// TIA Portal V17 export
// export: Created 2025-03-05T08:01:54.8682733Z, ExportSetting WithDefaults, DisplayName Totally Integrated Automation Portal, DisplayVersion V17 Update 8, DisplayName TIA Portal Openness, DisplayVersion V17 Update 8, DisplayName TIA Portal Version Control Interface, DisplayVersion V17, DisplayName SINAMICS Startdrive Advanced, DisplayVersion V17 SP2, DisplayName SINAMICS Startdrive G110M, G120, G120C, G120D, G120P, G115D, DisplayVersion V17 SP2, DisplayName SINAMICS Startdrive G130, G150, S120, S150, SINAMICS MV, S210, DisplayVersion V17 SP2, DisplayName STEP 7 Professional, DisplayVersion V17 Update 8, DisplayName SINUMERIK ONE STEP 7 Toolbox, DisplayVersion V17 Update 12, DisplayName SINUMERIK 840D sl STEP 7 Toolbox, DisplayVersion V17 Update 12, DisplayName STEP 7 Safety, DisplayVersion V17 Update 6, DisplayName WinCC Advanced, DisplayVersion V17 Update 8
TYPE "LBP_typeHMI"
TITLE = Operator panel signals / Señales panel de mando / Bedienfeld-Signale
// User data type for block LBP_HMI [DB19] / Tipo de dato de usuario para bloque LBP_HMI [DB19] / Anwender-Datentyp für Baustein LBP_HMI [DB19]
// stored: IsFailsafeCompliant false
   STRUCT
      A_SCLight : Bool;   // Bildschirm hell / Screen light / Pantalla luminosa
      A_SCDark : Bool;   // Bildschirm Abdunkelung / Screen darkening / Atenuación pantalla
      A_KeyDisable : Bool;   // Taste deaktivieren / Key disable / Desactivar tecla
      A_ClearCanAl : Bool;   // Abbruch-Alarme löschen / Clear cancel alarms / Borrar alarmas de cancelación
      A_ClearRecAl : Bool;   // Rückruf-Alarme löschen / Clear recall alarms / Borrar alarmas de rellamada
      f0_5 : Bool;
      A_SafeActionLog : Bool;   // Flankenwechsel 0 → 1: ACTION.COM nach CRASH.COM speichern / Edge change 0 → 1: Save ACTION.COM to CRASH.COM / Cambio de flanco 0 → 1: guardar ACTION.COM a CRASH.COM
      A_ActWCS : Bool;   // Istwert in WCS 0=MCS / Actual value in WCS 0=MCS / Valor real en WCS 0=MCS
      A_PLCExtViewerReject : Bool;   // Externen Viewer ablehnen / External viewer reject / Rechazar visualizador externo
      A_PLCExtViewerMode : Bool;   // Externer Viewer-Modus / External viewer mode / Modo de visualizador externo
      f1_2 : Bool;
      f1_3 : Bool;
      f1_4 : Bool;
      f1_5 : Bool;
      f1_6 : Bool;
      f1_7 : Bool;
      A_1stError1 : Word;   // 1. Fehler HIGRAPH / 1st error HIGRAPH / 1.er error HIGRAPH
      A_1stError2 : Word;   // 1. Fehler HIGRAPH / 1st error HIGRAPH / 1.er error HIGRAPH
      A_ASpi1percent : Byte;   // Analogspindel 1: / Analog spindle 1: / Cabezal analógico 1:
      A_ASpi2percent : Byte;
      A_MCPChan : Byte;
      A_OEM1 : Bool;
      A_OEM2 : Bool;
      A_AToolMeas : Bool;   // AutoToolMeasure
      f9_3 : Bool;
      f9_4 : Bool;
      f9_5 : Bool;
      f9_6 : Bool;
      f9_7 : Bool;
      A_Hardkey : Byte;   // PLC Hardkeys / PLC hardkeys / Pulsadores de función PLC
      f11 : Byte;   // Reserviert für Hardkeys / Reserved for hardkeys / Reservado para pulsadores de función
      f12_0 : Bool;
      f12_1 : Bool;
      A_COM2 : Bool;
      A_COM1 : Bool;
      A_V24stop : Bool;
      A_V24ext : Bool;
      A_V24off : Bool;
      A_V24on : Bool;
      A_TeachDisable : Bool;
      f13_1 : Bool;
      f13_2 : Bool;
      f13_3 : Bool;
      f13_4 : Bool;
      A_PPdeload : Bool;
      A_PPload : Bool;
      A_PPsel : Bool;
      A_V24Index1 : Byte;
      A_V24Index2 : Byte;
      A_V24NoFile1 : Byte;
      A_V24NoFile2 : Byte;
      A_res18 : Byte;
      A_res19 : Byte;   // Meldungszähler / Message counter / Contador de avisos
      f20_0 : Bool;
      E_SCDark : Bool;   // Bildschirm Abdunkelung / Screen darkening / Atenuación pantalla
      E_Cancel : Bool;   // Abbruch / Cancel / Cancelación
      E_CanCleared : Bool;   // Abbruch-Alarme gelöscht / Cancel alarms cleared / Alarmas de cancelación borradas
      E_RecCleared : Bool;   // Rückruf-Alarme gelöscht / Recall alarms cleared / Alarmas de rellamada borradas
      f20_5 : Bool;   // res. Sprache / res. language / Lenguaje res.
      E_SimActiv : Bool;   // Simulation aktiv / Simulation active / Simulación activa
      E_ActWCS : Bool;   // Umschaltung MCS/WCS 0=MCS / Switchover MCS/WCS 0=MCS / Conmutación MCS/WCS 0=MCS
      E_ActivWA : Byte;
      E_Chan : Byte;   // Kanal angezeigt / Channel displayed / Canal mostrado
      E_KeybHandl : Bool;   // Tastatur Handhabung / Keyboard handling / Manejo del teclado
      E_DataTransf : Bool;   // Datenübertragung aktiv / Data transfer active / Transferencia de datos activa
      E_DisplChange : Bool;   // Display Änderung / Display change / Cambio de visualización
      f23_3 : Bool;
      f23_4 : Bool;
      f23_5 : Bool;
      f23_6 : Bool;
      f23_7 : Bool;
      E_ScreenNo : Word;
      E_res26_0 : Bool;   // Reserviert / Reserved / Reservado
      E_PPOK : Bool;   // Teileprogramm-Status OK / Part program status OK / Estado programa de pieza OK
      E_PPErr : Bool;   // Teileprogramm Statusfehler / Part program status error / Estado programa de pieza error
      E_PPAct : Bool;   // Teileprogramm-Status aktiv / Part program status active / Estado programa de pieza activo
      f26_4 : Bool;   // Reserviert / Reserved / Reservado
      E_PPdeload : Bool;   // Teileprogramm-Status wird entladen / Part program status deloading / Estado programa de pieza en descarga
      E_PPload : Bool;   // Teileprogramm-Status wird geladen / Part program status loading / Estado programa de pieza en carga
      E_PPsel : Bool;   // Teileprogramm-Status wird ausgewählt / Part program status selecting / Estado programa de pieza se selecciona
      E_PPError : Byte;   // Teileprogramm Statusfehler / Part program status error / Estado programa de pieza error
      A_PictNo : Int;
      A_PictOn : Bool;
      A_PictOff : Bool;
      f30_2 : Bool;
      f30_3 : Bool;
      f30_4 : Bool;
      f30_5 : Bool;
      f30_6 : Bool;
      f30_7 : Bool;
      E_PictOK : Bool;
      E_PictOn : Bool;
      E_PictAct : Bool;
      E_PictOff : Bool;
      E_PictErr : Bool;
      f31_5 : Bool;
      f31_6 : Bool;
      E_NotAct : Bool;
      A_FuncNo : Byte;
      A_Par1 : Byte;
      A_Par2 : Byte;
      A_Par3 : Byte;
      E_FuncErr : Byte;
      f37 : Byte;
      f38 : Byte;
      f39 : Byte;
      res40 : Array[0..9] of Byte;
      MMC2 : Struct
         A_SCLight : Bool;   // Bildschirm hell / Screen light / Pantalla luminosa
         A_SCDark : Bool;   // Bildschirm Abdunkelung / Screen darkening / Atenuación pantalla
         A_KeyDisable : Bool;   // Taste deaktivieren / Key disable / Desactivar tecla
         A_ClearCanAl : Bool;   // Abbruch-Alarme löschen / Clear cancel alarms / Borrar alarmas de cancelación
         A_ClearRecAl : Bool;   // Rückruf-Alarme löschen / Clear recall alarms / Borrar alarmas de rellamada
         f0_5 : Bool;
         f0_6 : Bool;
         A_ActWCS : Bool;   // Istwert in WCS 0=MCS / Actual value in WCS 0=MCS / Valor real en WCS 0=MCS
         A_PLCExtViewerReject : Bool;   // Externen Viewer ablehnen / External viewer reject / Rechazar visualizador externo
         A_PLCExtViewerMode : Bool;   // Externer Viewer-Modus / External viewer mode / Modo de visualizador externo
         f1_2 : Bool;
         f1_3 : Bool;
         f1_4 : Bool;
         f1_5 : Bool;
         f1_6 : Bool;
         f1_7 : Bool;
         A_1stError1 : Word;   // 1. Fehler HIGRAPH / 1st error HIGRAPH / 1.er error HIGRAPH
         A_1stError2 : Word;   // 1. Fehler HIGRAPH / 1st error HIGRAPH / 1.er error HIGRAPH
         A_ASpi1percent : Byte;   // Analogspindel 1: / Analog spindle 1: / Cabezal analógico 1:
         A_ASpi2percent : Byte;
         A_MCPChan : Byte;
         A_OEM1 : Bool;
         A_OEM2 : Bool;
         A_AToolMeas : Bool;   // AutoToolMeasure
         f9_3 : Bool;
         f9_4 : Bool;
         f9_5 : Bool;
         f9_6 : Bool;
         f9_7 : Bool;
         A_Hardkey : Byte;   // PLC Hardkeys / PLC hardkeys / Pulsadores de función PLC
         f11 : Byte;   // Reserviert für Hardkeys / Reserved for hardkeys / Reservado para pulsadores de función
         f12_0 : Bool;
         f12_1 : Bool;
         A_COM2 : Bool;
         A_COM1 : Bool;
         A_V24stop : Bool;
         A_V24ext : Bool;
         A_V24off : Bool;
         A_V24on : Bool;
         A_TeachDisable : Bool;
         f13_1 : Bool;
         f13_2 : Bool;
         f13_3 : Bool;
         f13_4 : Bool;
         A_PPdeload : Bool;
         A_PPload : Bool;
         A_PPsel : Bool;
         A_V24Index1 : Byte;
         A_V24Index2 : Byte;
         A_V24NoFile1 : Byte;
         A_V24NoFile2 : Byte;
         A_res18 : Byte;
         A_res19 : Byte;   // Meldungszähler / Message counter / Contador de avisos
         f20_0 : Bool;
         E_SCDark : Bool;   // Bildschirm Abdunkelung / Screen darkening / Atenuación pantalla
         E_Cancel : Bool;   // Abbruch / Cancel / Cancelación
         E_CanCleared : Bool;   // Abbruch-Alarme gelöscht / Cancel alarms cleared / Alarmas de cancelación borradas
         E_RecCleared : Bool;   // Rückruf-Alarme gelöscht / Recall alarms cleared / Alarmas de rellamada borradas
         f20_5 : Bool;   // res. Sprache / res. language / Lenguaje res.
         E_SimActiv : Bool;   // Simulation aktiv / Simulation active / Simulación activa
         E_ActWCS : Bool;   // Umschaltung MCS/WCS 0=MCS / Switchover MCS/WCS 0=MCS / Conmutación MCS/WCS 0=MCS
         E_ActivWA : Byte;
         E_Chan : Byte;   // Kanal angezeigt / Channel displayed / Canal mostrado
         E_KeybHandl : Bool;   // Tastatur Handhabung / Keyboard handling / Manejo del teclado
         E_DataTransf : Bool;   // Datenübertragung aktiv / Data transfer active / Transferencia de datos activa
         E_DisplChange : Bool;   // Display Änderung / Display change / Cambio de visualización
         f23_3 : Bool;
         f23_4 : Bool;
         f23_5 : Bool;
         f23_6 : Bool;
         f23_7 : Bool;
         E_ScreenNo : Word;
         E_res26_0 : Bool;   // Reserviert / Reserved / Reservado
         E_PPOK : Bool;   // Teileprogramm-Status OK / Part program status OK / Estado programa de pieza OK
         E_PPErr : Bool;   // Teileprogramm Statusfehler / Part program status error / Estado programa de pieza error
         E_PPAct : Bool;   // Teileprogramm-Status aktiv / Part program status active / Estado programa de pieza activo
         f26_4 : Bool;   // Reserviert / Reserved / Reservado
         E_PPdeload : Bool;   // Teileprogramm-Status wird entladen / Part program status deloading / Estado programa de pieza en descarga
         E_PPload : Bool;   // Teileprogramm-Status wird geladen / Part program status loading / Estado programa de pieza en carga
         E_PPsel : Bool;   // Teileprogramm-Status wird ausgewählt / Part program status selecting / Estado programa de pieza se selecciona
         E_PPError : Byte;   // Teileprogramm Statusfehler / Part program status error / Estado programa de pieza error
         A_PictNo : Int;
         A_PictOn : Bool;
         A_PictOff : Bool;
         f30_2 : Bool;
         f30_3 : Bool;
         f30_4 : Bool;
         f30_5 : Bool;
         f30_6 : Bool;
         f30_7 : Bool;
         E_PictOK : Bool;
         E_PictOn : Bool;
         E_PictAct : Bool;
         E_PictOff : Bool;
         E_PictErr : Bool;
         f31_5 : Bool;
         f31_6 : Bool;
         E_NotAct : Bool;
         A_FuncNo : Byte;
         A_Par1 : Byte;
         A_Par2 : Byte;
         A_Par3 : Byte;
         E_FuncErr : Byte;
         f37 : Byte;
         f38 : Byte;
         f39 : Byte;
         res40 : Array[0..9] of Byte;
      END_STRUCT;
      ONL_REQUEST : Word;
      ONL_CONFIRM : Word;
      PAR_CLIENT_IDENT : Word;
      PAR_MMC_TYP : Byte;
      PAR_MSTT_ADR : Byte;
      PAR_STATUS : Byte;
      PAR_Z_INFO : Byte;
      MtoNAlive : Word;
      f112 : Byte;
      ParOpKeyAdr : Byte;
      ParTcuIndex : Byte;
      f115 : Byte;
      Tcu1KeyAdr : Byte;
      Tcu2KeyAdr : Byte;
      Tcu1Index : Byte;
      Tcu2Index : Byte;
      MMC1_CLIENT_IDENT : Word;
      MMC1_TYP : Byte;
      MMC1_MSTT_ADR : Byte;
      MMC1_STATUS : Byte;
      MMC1_Z_INFO : Byte;
      MMC1_SHIFT_LOCK : Bool;
      MMC1_MSTT_SHIFT_LOCK : Bool;
      MMC1_ACTIVE_REQ : Bool;
      MMC1_ACTIVE_PERM : Bool;
      MMC1_ACTIVE_CHANGED : Bool;
      MMC1_CHANGED_DENIED : Bool;
      MMC1_TCU_SHIFT_LOCK : Bool;
      f127 : Byte;
      MMC1_TRANS_DB : Word;
      MMC2_CLIENT_IDENT : Word;
      MMC2_TYP : Byte;
      MMC2_MSTT_ADR : Byte;
      MMC2_STATUS : Byte;
      MMC2_Z_INFO : Byte;
      MMC2_SHIFT_LOCK : Bool;
      MMC2_MSTT_SHIFT_LOCK : Bool;
      MMC2_ACTIVE_REQ : Bool;
      MMC2_ACTIVE_PERM : Bool;
      MMC2_ACTIVE_CHANGED : Bool;
      MMC2_CHANGED_DENIED : Bool;
      MMC2_TCU_SHIFT_LOCK : Bool;
      f137 : Byte;
      MMC2_TRANS_DB : Word;
      A_Subtype : Int;   // Für Codeträger Eingabe aus PLC / For code carrier Input from PLC / Para portador codificado Entrada desde PLC
      A_Duplo : Int;
      A_Ident : String[32];
      A_Tnumber : Int;
      A_MagazinePlace : Int;
      A_MagazinePlaceType : Int;
      A_ToolSize_Upper : Byte;
      A_ToolSize_Down : Byte;
      A_ToolSize_Left : Byte;
      A_ToolSize_Right : Byte;
      A_Channel : Byte;
      A_LoadingPlace : Byte;
      A_Magazine : Int;
      A_Unit : Byte;
      A_NCU_Index : Byte;
      A_FileIndex : Int;
      A_ActiveEnable : Bool;
      A_Override : Bool;
      A_LoadTool : Bool;
      A_DeleteTool : Bool;
      E_Subtype : Int;   // Für Codeträger Ausgabe an PLC / For code carrier Output to PLC / Para portador codificado Salida a PLC
      E_Duplo : Int;
      E_Ident : String[32];
      E_Tnumber : Int;
      E_ToolState : Int;
      E_MagazinePlaceType : Int;
      E_ToolSize_Upper : Byte;
      E_ToolSize_Down : Byte;
      E_ToolSize_Left : Byte;
      E_ToolSize_Right : Byte;
      E_Magazine : Int;
      E_MagazinePlace : Int;
      A_ReqMMC1 : Bool;   // Für Codeträger MMC-Schnittstelle 1 anfordern / For code carrier Request MMC-Interface1 / Para portador codificado Solicitar interfaz MMC 1
      A_ReqMMC2 : Bool;   // Für Codeträger MMC-Schnittstelle 2 anfordern / For code carrier Request MMC-Interface2 / Para portador codificado Solicitar interfaz MMC 2
      A_K_Code : Byte;
      E_Done : Bool;
      E_Error : Bool;
      E_Active : Bool;
      f252_3 : Bool;
      f252_4 : Bool;
      f252_5 : Bool;
      f252_6 : Bool;
      E_Ident_Ready : Bool;
      E_K_CodeError : Byte;   // Identifizieren für Error_Code / Identify for Error_Code / Identificar para Error_Code
      E_Error_Code : Int;
      E_Req : Bool;   // Für Positionierung / For Positioning / Para posicionamiento
      f257 : Byte;
      A_Done : Bool;
      A_Error : Bool;
      A_Active : Bool;
      f258_3 : Bool;
      f258_4 : Bool;
      f258_5 : Bool;
      f258_6 : Bool;
      f258_7 : Bool;
      E_TDC_Read : Bool;
      E_TDC_Write : Bool;
      E_TDC_Cancel : Bool;
      E_TDC_Read_before_Write : Bool;
      f259_4 : Bool;
      f259_5 : Bool;
      f259_6 : Bool;
      f259_7 : Bool;
      A_Error_Code : Int;
      E_PMagazine : Int;
      E_PMagazinePlace : Int;
      E_PTnumber : Int;   // TPM-Daten / TPM data / Datos TPM
      A_TPMStatus : Int;
      A_TPMCounter : Array[1..32] of DInt;
      A_HWeelSimOvr : Byte;
      f399 : Byte;
      A_SimOvr : Int;   // Simulation Override / Simulation override / Corregir simulación
      A_SimState : Int;   // Simulationszustand / Simulation state / Estado simulación
      E_HmiUserKey : Array[1..64] of Bool;   // HMI Anwender-Tasten für HMI-Seitenmonitor / HMI user keys for HMI sidescreen / HMI teclas de usuario para Sidescreen del HMI
      A_HmiUserLed : Array[1..64] of Bool;   // LEDs für Anwender-Tasten für HMI Seitenmonitor / LEDs to the user keys for HMI sidescreen / LED para teclas de usuario para Sidescreen del HMI
      A_DisableHmiUserKey : Array[1..64] of Bool;   // Anwender-Tasten für HMI-Seitenmonitor deaktivieren / Disable user keys for HMI sidescreen / Desactivar teclas de usuario para Sidescreen del HMI
   END_STRUCT;
END_TYPE
